(*
	Return sign of input value
*)
{attribute 'hide_all_locals'}
FUNCTION F_Sign : REAL
VAR_INPUT
	fValue 	: REAL;
END_VAR

IF (fValue >= 0) THEN
	F_Sign := 1;
ELSE
	F_Sign := -1;	
END_IF

END_FUNCTION

(* stored: Version 1.1.0.1, ProductVersion 3.1.4024.12
   POU F_Sign: Id {60b99345-8786-0015-08b7-72f2bf3aa665}, SpecialFunc None *)
